% RSLogix 500 project PLC_1_L4-2.RSS, saved by version 12.00.00.00 %
PROJECT "UNTITLED"    % processor: Bul.1763 MicroLogix 1100 Series B %

PROGRAM FILES
  LAD 2   2 rungs

DATA FILES
  O0 OUTPUT  5 elements
  I1 INPUT  6 elements
  S2 STATUS  66 elements
  B3 BINARY  1 elements
  T4 TIMER  1 elements
  C5 COUNTER  1 elements
  R6 CONTROL  1 elements
  N7 INTEGER  1 elements
  F8 FLOAT  1 elements

LADDER 2
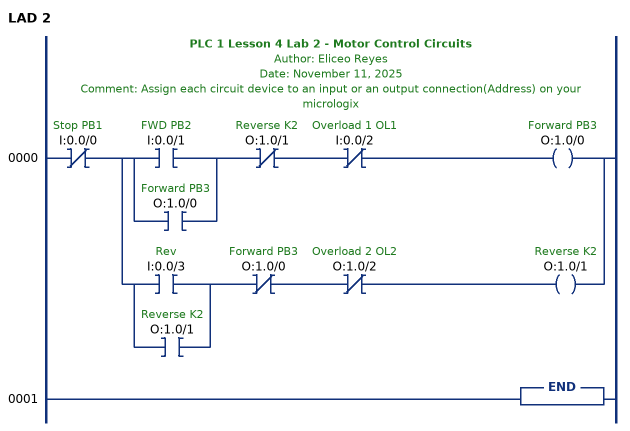
% Rung: 0 %
% TITLE: PLC 1 Lesson 4 Lab 2 - Motor Control Circuits %
% Author: Eliceo Reyes
% Date: November 11, 2025
% Comment: Assign each circuit device to an input or an output connection(Address) on your micrologix %
SOR XIO I:0.0/0 BST BST XIC I:0.0/1 NXB XIC O:1.0/0 BND XIO O:1.0/1 XIO I:0.0/2 OTE O:1.0/0 NXB BST XIC I:0.0/3 NXB XIC O:1.0/1 BND XIO O:1.0/0 XIO O:1.0/2 OTE O:1.0/1 BND EOR
%   I:0.0/0  PB1  "Stop" %
%   I:0.0/1  PB2  "FWD" %
%   O:1.0/0  PB3  "Forward" %
%   O:1.0/1  K2  "Reverse" %
%   I:0.0/2  OL1  "Overload 1" %
%   I:0.0/3  "Rev" %
%   O:1.0/2  OL2  "Overload 2" %
% Rung: 1 %
SOR END EOR
